// TIA Portal project "tank_automation" (V17)
// Vorlageprojekt für das Buch mit Zielsystem S7-1200

(* hardware
DEVICE "HMI_1"  KTP700 Basic PN
   slot 0: "HMI_1"  KTP700 Basic PN  6AV2 123-2GB03-0AX0  17.0.0.0
   slot 1: "HMI_RT_1"  KTP700 Basic PN  6AV2 123-2GB03-0AX0  17.0.0.0
   slot 5: "HMI_1.IE_CP_1"  PROFINET Interface  17.0.0.0
      slot 1: "PROFINET Interface_1"  PROFINET Interface
         slot 1: "Port_1"  Port
DEVICE "S7-1200 station_1"  S7-1200 Station
   slot 0: "Rack_0"  S7-1200 Rack  Rack  V1.0
   slot 1: "PLC_2"  CPU 1214C DC/DC/DC  6ES7 214-1AG40-0XB0  V4.5
   slot 2: "AQ 2x14BIT_1"  SM 1232 AQ2  6ES7 232-4HB32-0XB0  V2.1
*)

// ===== PLC "PLC_2"  CPU 1214C DC/DC/DC =====

VAR_GLOBAL   // PLC tag table "Default tag table"
   "Level Meter" AT %IW30 : Int;
   "HMI Filling Speed Up" AT %M20.0 : Bool;
   "Tag_5" AT %M20.1 : Bool;
   "Filling Speed Memory" AT %MW30 : Int;
   "HMI Filling Speed Down" AT %M20.2 : Bool;
   "Tag_6" AT %M20.3 : Bool;
   "Fill Valve" AT %QW30 : Int;
   "Level Meter Percentage" AT %MD10 : Real;
   "Tank Level Value" AT %MD14 : Real;
   "Pump" AT %Q0.0 : Bool;
   "HMI Discharge Speed Up" AT %M20.4 : Bool;
   "Tag_2" AT %M20.5 : Bool;
   "Discharge Speed Memory" AT %MW32 : Int;
   "HMI Discharge Speed Down" AT %M20.6 : Bool;
   "Tag_3" AT %M20.7 : Bool;
   "Discharge Valve" AT %QW32 : Int;
   "HMI Lever" AT %M40.0 : Bool;
END_VAR

DATA_BLOCK "DB_Tank"   // DB1
{ S7_Optimized_Access := 'TRUE' }
VERSION : 0.1
   VAR
      Level_RAW_Buffer : Int;
      Level_Percent : Real;
      Level_Value : Real;
   END_VAR
BEGIN
END_DATA_BLOCK

FUNCTION "Manual Operation" : Void   // FC1, LAD
{ S7_Optimized_Access := 'TRUE' }
VERSION : 0.1
   VAR_TEMP   // added for the SCL form of the ladder/FBD networks
      _w1 : Bool;
      _w2 : Bool;
   END_VAR
BEGIN

REGION Network 1
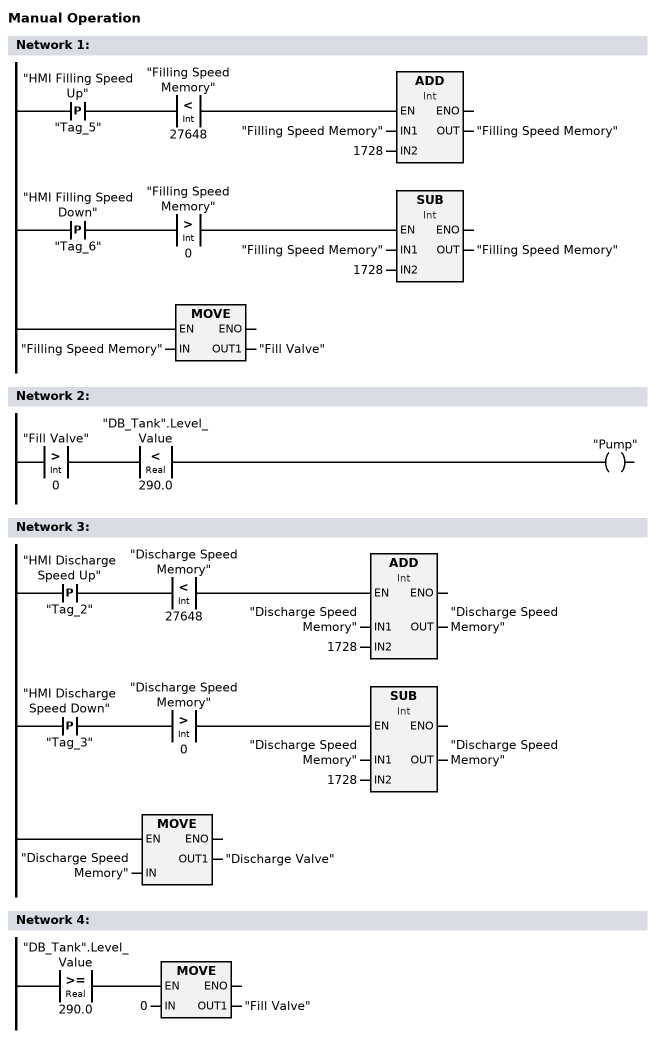
   RUNG wire#powerrail
      P_Contact(operand := "HMI Filling Speed Up", bit := "Tag_5")
      { S7_Templates := "SrcType := Int" } LT_Contact(in1 := "Filling Speed Memory", in2 := 27648)
      { S7_Templates := "SrcType := Int" } Add(in1 := "Filling Speed Memory", in2 := 1728, out => "Filling Speed Memory")
   END_RUNG
   RUNG wire#powerrail
      P_Contact(operand := "HMI Filling Speed Down", bit := "Tag_6")
      { S7_Templates := "SrcType := Int" } GT_Contact(in1 := "Filling Speed Memory", in2 := 0)
      { S7_Templates := "SrcType := Int" } Sub(in1 := "Filling Speed Memory", in2 := 1728, out => "Filling Speed Memory")
   END_RUNG
   RUNG wire#powerrail
      Move(in := "Filling Speed Memory", out1 => "Fill Valve")
   END_RUNG
   // the same network as SCL:
   #_w1 := "HMI Filling Speed Up" AND NOT "Tag_5";   // rising edge of "HMI Filling Speed Up"
   "Tag_5" := "HMI Filling Speed Up";
   IF #_w1 AND ("Filling Speed Memory" < 27648) THEN
       "Filling Speed Memory" := "Filling Speed Memory" + 1728;
   END_IF;
   #_w2 := "HMI Filling Speed Down" AND NOT "Tag_6";   // rising edge of "HMI Filling Speed Down"
   "Tag_6" := "HMI Filling Speed Down";
   IF #_w2 AND ("Filling Speed Memory" > 0) THEN
       "Filling Speed Memory" := "Filling Speed Memory" - 1728;
   END_IF;
   "Fill Valve" := "Filling Speed Memory";
END_REGION

REGION Network 2
   RUNG wire#powerrail
      { S7_Templates := "SrcType := Int" } GT_Contact(in1 := "Fill Valve", in2 := 0)
      { S7_Templates := "SrcType := Real" } LT_Contact(in1 := "DB_Tank".Level_Value, in2 := 290.0)
      Coil( "Pump" )
   END_RUNG
   // the same network as SCL:
   "Pump" := ("Fill Valve" > 0) AND ("DB_Tank".Level_Value < 290.0);
END_REGION

REGION Network 3
   RUNG wire#powerrail
      P_Contact(operand := "HMI Discharge Speed Up", bit := "Tag_2")
      { S7_Templates := "SrcType := Int" } LT_Contact(in1 := "Discharge Speed Memory", in2 := 27648)
      { S7_Templates := "SrcType := Int" } Add(in1 := "Discharge Speed Memory", in2 := 1728, out => "Discharge Speed Memory")
   END_RUNG
   RUNG wire#powerrail
      P_Contact(operand := "HMI Discharge Speed Down", bit := "Tag_3")
      { S7_Templates := "SrcType := Int" } GT_Contact(in1 := "Discharge Speed Memory", in2 := 0)
      { S7_Templates := "SrcType := Int" } Sub(in1 := "Discharge Speed Memory", in2 := 1728, out => "Discharge Speed Memory")
   END_RUNG
   RUNG wire#powerrail
      Move(in := "Discharge Speed Memory", out1 => "Discharge Valve")
   END_RUNG
   // the same network as SCL:
   #_w1 := "HMI Discharge Speed Up" AND NOT "Tag_2";   // rising edge of "HMI Discharge Speed Up"
   "Tag_2" := "HMI Discharge Speed Up";
   IF #_w1 AND ("Discharge Speed Memory" < 27648) THEN
       "Discharge Speed Memory" := "Discharge Speed Memory" + 1728;
   END_IF;
   #_w2 := "HMI Discharge Speed Down" AND NOT "Tag_3";   // rising edge of "HMI Discharge Speed Down"
   "Tag_3" := "HMI Discharge Speed Down";
   IF #_w2 AND ("Discharge Speed Memory" > 0) THEN
       "Discharge Speed Memory" := "Discharge Speed Memory" - 1728;
   END_IF;
   "Discharge Valve" := "Discharge Speed Memory";
END_REGION

REGION Network 4
   RUNG wire#powerrail
      { S7_Templates := "SrcType := Real" } GE_Contact(in1 := "DB_Tank".Level_Value, in2 := 290.0)
      Move(in := 0, out1 => "Fill Valve")
   END_RUNG
   // the same network as SCL:
   IF "DB_Tank".Level_Value >= 290.0 THEN "Fill Valve" := 0; END_IF;
END_REGION
END_FUNCTION

FUNCTION "Automatic Operation" : Void   // FC2, LAD
{ S7_Optimized_Access := 'TRUE' }
VERSION : 0.1
BEGIN

REGION Network 1
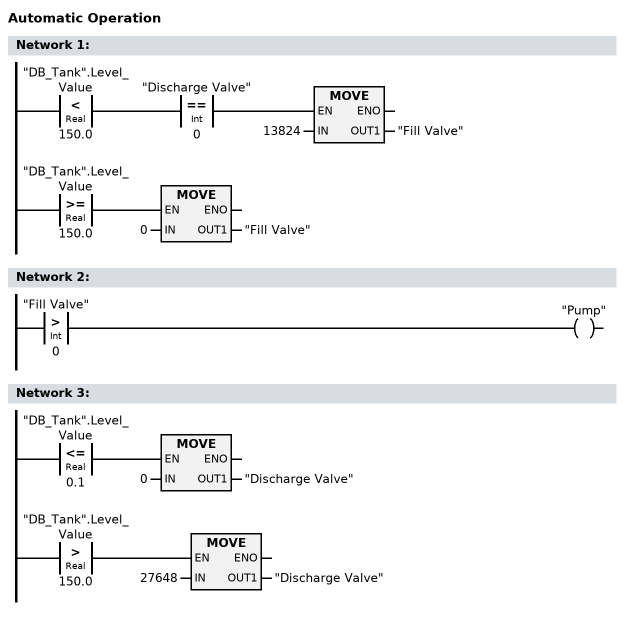
   RUNG wire#powerrail
      { S7_Templates := "SrcType := Real" } LT_Contact(in1 := "DB_Tank".Level_Value, in2 := 150.0)
      { S7_Templates := "SrcType := Int" } EQ_Contact(in1 := "Discharge Valve", in2 := 0)
      Move(in := 13824, out1 => "Fill Valve")
   END_RUNG
   RUNG wire#powerrail
      { S7_Templates := "SrcType := Real" } GE_Contact(in1 := "DB_Tank".Level_Value, in2 := 150.0)
      Move(in := 0, out1 => "Fill Valve")
   END_RUNG
   // the same network as SCL:
   IF ("DB_Tank".Level_Value < 150.0) AND ("Discharge Valve" = 0) THEN "Fill Valve" := 13824; END_IF;
   IF "DB_Tank".Level_Value >= 150.0 THEN "Fill Valve" := 0; END_IF;
END_REGION

REGION Network 2
   RUNG wire#powerrail
      { S7_Templates := "SrcType := Int" } GT_Contact(in1 := "Fill Valve", in2 := 0)
      Coil( "Pump" )
   END_RUNG
   // the same network as SCL:
   "Pump" := "Fill Valve" > 0;
END_REGION

REGION Network 3
   RUNG wire#powerrail
      { S7_Templates := "SrcType := Real" } LE_Contact(in1 := "DB_Tank".Level_Value, in2 := 0.1)
      Move(in := 0, out1 => "Discharge Valve")
   END_RUNG
   RUNG wire#powerrail
      { S7_Templates := "SrcType := Real" } GT_Contact(in1 := "DB_Tank".Level_Value, in2 := 150.0)
      Move(in := 27648, out1 => "Discharge Valve")
   END_RUNG
   // the same network as SCL:
   IF "DB_Tank".Level_Value <= 0.1 THEN "Discharge Valve" := 0; END_IF;
   IF "DB_Tank".Level_Value > 150.0 THEN "Discharge Valve" := 27648; END_IF;
END_REGION
END_FUNCTION

FUNCTION "MHJ-PLC-Lab-Function-S71200" : Void   // FC9000, SCL
{ S7_Optimized_Access := 'TRUE' }
VERSION : 0.1
   VAR_TEMP
      rdTimeReturn : Int;
      outputTime : DTL;
      SyncVal : Byte;
      forVal : Int;
      forVal_2 : Int;
      Value : Byte;
   END_VAR
   VAR CONSTANT
      CompVal : Byte := 16#34;
      Value_01 : Byte := 16#11;
      Value_01_DW : DWord := 16#A165_D992;
      Value_02_DW : DWord := 16#58BE_4401;
   END_VAR
BEGIN

   #Value:=PEEK(area := 16#82,
        dbNumber := 0,
        byteOffset := 511);
   #Value := #Value + 1;

   POKE(area := 16#82,
        dbNumber := 0,
        byteOffset := 511,
        value := #Value);

   POKE(area:=16#81,
        dbNumber:=0,
        byteOffset:=1016,
        value:=#Value_01_DW);
   POKE(area := 16#81,
        dbNumber := 0,
        byteOffset := 1020,
        value := #Value_02_DW);

   POKE(area := 16#81,
        dbNumber := 0,
        byteOffset := 511,
        value := B#16#00);

   FOR #forVal := 0 TO 120 DO
       FOR #forVal_2:=0 TO 10 DO
           #rdTimeReturn:=RD_SYS_T(#outputTime);
           #rdTimeReturn := WR_SYS_T(#outputTime);
           #rdTimeReturn := RD_SYS_T(#outputTime);
           #rdTimeReturn := WR_SYS_T(#outputTime);
       END_FOR;
       #SyncVal:= PEEK(area := 16#81,
                      dbNumber := 0,
                      byteOffset := 511);
       IF #SyncVal = #CompVal THEN
          GOTO M_1;
       END_IF;
   END_FOR;
   RETURN;

   M_1:
   POKE(area := 16#81,
        dbNumber := 0,
        byteOffset := 511,
        value := B#16#0);
END_FUNCTION

ORGANIZATION_BLOCK "Main"   // OB1, LAD, ProgramCycle
TITLE = "Main Program Sweep (Cycle)"
{ S7_Optimized_Access := 'TRUE' }
VERSION : 0.1
   VAR_INPUT
      Initial_Call : Bool;   // Initial call of this OB
      Remanence : Bool;   // =True, if remanent data are available
   END_VAR
BEGIN

REGION Network 1: Konnektierungsbaustein für PLC-Lab
   // Im Netzwerk 1 wird der Konnektierungsbaustein für PLC-Lab aufgerufen.
   // Dieser Aufruf darf nicht entfernt werden!
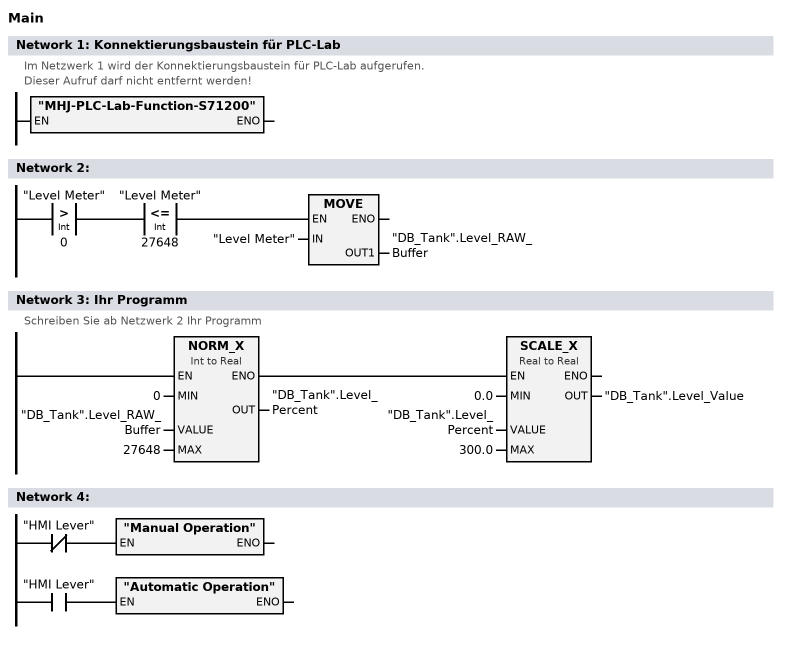
   RUNG wire#powerrail
      "MHJ-PLC-Lab-Function-S71200"()
   END_RUNG
   // the same network as SCL:
   "MHJ-PLC-Lab-Function-S71200"();
END_REGION

REGION Network 2
   RUNG wire#powerrail
      { S7_Templates := "SrcType := Int" } GT_Contact(in1 := "Level Meter", in2 := 0)
      { S7_Templates := "SrcType := Int" } LE_Contact(in1 := "Level Meter", in2 := 27648)
      Move(in := "Level Meter", out1 => "DB_Tank".Level_RAW_Buffer)
   END_RUNG
   // the same network as SCL:
   IF ("Level Meter" > 0) AND ("Level Meter" <= 27648) THEN
       "DB_Tank".Level_RAW_Buffer := "Level Meter";
   END_IF;
END_REGION

REGION Network 3: Ihr Programm
   // Schreiben Sie ab Netzwerk 2 Ihr Programm
   RUNG wire#powerrail
      { S7_Templates := "[SrcType := Int, DestType := Real]" } Normalize(min := 0, value := "DB_Tank".Level_RAW_Buffer, max := 27648, out => "DB_Tank".Level_Percent)
      { S7_Templates := "[SrcType := Real, DestType := Real]" } Scale(min := 0.0, value := "DB_Tank".Level_Percent, max := 300.0, out => "DB_Tank".Level_Value)
   END_RUNG
   // the same network as SCL:
   "DB_Tank".Level_Percent := NORM_X(MIN := 0, VALUE := "DB_Tank".Level_RAW_Buffer, MAX := 27648);
   "DB_Tank".Level_Value := SCALE_X(MIN := 0.0, VALUE := "DB_Tank".Level_Percent, MAX := 300.0);
END_REGION

REGION Network 4
   RUNG wire#powerrail
      I_Contact( "HMI Lever" )
      "Manual Operation"()
   END_RUNG
   RUNG wire#powerrail
      Contact( "HMI Lever" )
      "Automatic Operation"()
   END_RUNG
   // the same network as SCL:
   IF NOT "HMI Lever" THEN "Manual Operation"(); END_IF;
   IF "HMI Lever" THEN "Automatic Operation"(); END_IF;
END_REGION
END_ORGANIZATION_BLOCK

(* ===== HMI "HMI_RT_1" =====
system functions are stored by id; their names below are inferred from use
connection "HMI_Connection_2": ETHERNET, SMART_S7_1200_OMS

HMI tags "Default tag table"
   "HMI Lever" : Bool = PLC "HMI Lever" AT %M40.0, 1 s
   "Fill Valve" : Int = PLC "Fill Valve" AT %QW30, 1 s
   "Discharge Valve" : Int = PLC "Discharge Valve" AT %QW32, 1 s
   "Pump" : Bool = PLC Pump AT %Q0.0, 1 s
   "Tank Level Value" : Real = PLC "Tank Level Value" AT %MD14, 1 s
   "HMI Filling Speed Up" : Bool = PLC "HMI Filling Speed Up" AT %M20.0, 1 s
   "HMI Filling Speed Down" : Bool = PLC "HMI Filling Speed Down" AT %M20.2, 1 s
   "HMI Discharge Speed Up" : Bool = PLC "HMI Discharge Speed Up" AT %M20.4, 1 s
   "HMI Discharge Speed Down" : Bool = PLC "HMI Discharge Speed Down" AT %M20.6, 1 s
   "Filling Speed Memory" : Int = PLC "Filling Speed Memory" AT %MW30, 1 s
   "Discharge Speed Memory" : Int = PLC "Discharge Speed Memory" AT %MW32, 1 s
   "Data_block_1_Level_Value" : Real = PLC DB_Tank.Level_Value, 1 s

graphic list "Valve Graphics List": 0 'Graphic_16'; 1..27648 'Graphic_10'

graphic list "Pump Graphics List": 0 'Graphic_12'; 1 'Graphic_13'

screen "Root screen" 800x480, template "Template_1"
   TextField "Text field_1" at 328,19 size 133x29; Text 'TANK LEVEL'
   GraphicIOField "Graphic I/O field_1" at 403,110 size 60x55; PictureList "Valve Graphics List"
      ProcessValue <- "Fill Valve"
   GraphicIOField "Graphic I/O field_3" at 41,364 size 137x86; PictureList "Pump Graphics List"
      ProcessValue <- "Pump"
   GraphicView "Graphic view_2" at 175,384 size 145x43; Picture "Graphic_19"
   GraphicView "Graphic view_3" at 319,384 size 43x43; Picture "Graphic_20"
   GraphicView "Graphic view_5" at 319,168 size 43x218; Picture "Graphic_22"
   GraphicView "Graphic view_4" at 319,127 size 43x43; Picture "Graphic_23"
   GraphicView "Graphic view_6" at 361,127 size 48x43; Picture "Graphic_19"
   GraphicView "Graphic view_7" at 456,127 size 43x43; Picture "Graphic_24"
   GraphicIOField "Graphic I/O field_2" at 613,389 size 60x55; PictureList "Valve Graphics List"
      ProcessValue <- "Discharge Valve"
   GraphicView "Graphic view_8" at 571,406 size 48x43; Picture "Graphic_19"
   GraphicView "Graphic view_1" at 384,165 size 191x289; Picture "Graphic_14"
   GraphicView "Graphic view_9" at 666,406 size 134x43; Picture "Graphic_19"
   Bar "Bar_1" at 450,199 size 54x240; MinimumValue 0; MaximumValue 300
      ProcessValue <- "Data_block_1_Level_Value"
   Switch "Lever_Vertical_1" at 582,253 size 50x80; CaptionText 'Switch'; TextOff '0'; TextOn '1'; PictureOff "Lever_Vertical_1_Off_256c"; PictureOn "Lever_Vertical_1_On_256c"
      ProcessValue <- "HMI Lever"
   TextField "Text field_2" at 632,253 size 80x22; Text 'Automatic'
   TextField "Text field_3" at 632,309 size 59x22; Text 'Manual'
   Button "Button_1" at 50,180 size 55x50; TextOff 'Text'; PictureOff "Up_Arrow"
      on Press: SetBit("HMI Filling Speed Up")
      on Release: ResetBit("HMI Filling Speed Up")
   Button "Button_2" at 50,240 size 55x50; TextOff 'Text'; PictureOff "Down_Arrow"
      on Press: SetBit("HMI Filling Speed Down")
      on Release: ResetBit("HMI Filling Speed Down")
   TextField "Text field_4" at 16,140 size 128x23; Text 'FILLING SPEED'
   Button "Button_3" at 210,180 size 55x50; TextOff 'Text'; PictureOff "Up_Arrow"
      on Press: SetBit("HMI Discharge Speed Up")
      on Release: ResetBit("HMI Discharge Speed Up")
   Button "Button_4" at 210,240 size 55x50; TextOff 'Text'; PictureOff "Down_Arrow"
      on Press: SetBit("HMI Discharge Speed Down")
      on Release: ResetBit("HMI Discharge Speed Down")
   TextField "Text field_5" at 160,140 size 161x23; Text 'DISCHARGE SPEED'
   IOField "I/O field_1" at 45,300 size 64x32; FormatPattern 999
      ProcessValue <- "Filling Speed Memory"
   IOField "I/O field_2" at 205,300 size 64x32; FormatPattern 999
      ProcessValue <- "Discharge Speed Memory"
*)